{attribute 'qualified_only'}
{attribute 'strict'}
TYPE E_State :
(
	STATE_1_Listen,
	STATE_2_Accept,
	STATE_3_Receive,
	STATE_4_Send
);
END_TYPE

(* stored: Version 1.1.0.1, ProductVersion 3.1.4024.12
   DUT E_State: Id {949a7540-a87b-48ab-8e1d-061c13993609} *)
